# EPICS substitutions: iocBoot/iocFalconX1/1element.substitutions
file "$(DXP_SITORO)/db/dxpSystem.template" {
{P=dxpSITORO:, IO="@asyn(DXP1,0)"}
}

file "$(DXP_SITORO)/db/dxpMED.template" {
{P=dxpSITORO:, DETALL="@asyn(DXP1,1,1)"}
}

file "$(DXP_SITORO)/db/dxpMapping.template" {
{P=dxpSITORO:, IO="@asyn(DXP1,0)"}
}

# DXP parameters
file "$(DXP_SITORO)/db/dxpHighLevel.template"
{
pattern
{         P,       R,           IO}
{dxpSITORO:,    dxp1:,  "@asyn(DXP1,0,1)"}
}

# SCA parameters
file "$(DXP_SITORO)/db/dxpSCA.template"
{
pattern
{         P,       R,   N,        IO}
{dxpSITORO:,    dxp1:,  0, "@asyn(DXP1,0,1)"}
{dxpSITORO:,    dxp1:,  1, "@asyn(DXP1,0,1)"}
{dxpSITORO:,    dxp1:,  2, "@asyn(DXP1,0,1)"}
{dxpSITORO:,    dxp1:,  3, "@asyn(DXP1,0,1)"}
}

file "$(MCA)/db/simple_mca.db"
{
pattern
{         P,      M,       DTYP,               INP,  PREC,    CHANS}
{dxpSITORO:,   mca1,  "asynMCA",   "@asyn(DXP1,0)",     2,     2048}
}

file "$(ASYN)/db/asynRecord.db"
{
pattern
{       P,      R,  PORT,   ADDR,  IMAX,  OMAX}
{dxpSITORO:, Asyn,  DXP1,      0,    80,    80}
}
